PROGRAM CraneControl
VAR
	fbControlBox : FB_ControlBox; 
 	fbStatus : FB_Status;
	fbManualControl : FB_ManualControl; 
	bEnableManualControl : BOOL;
	fbAutomaticControl : FB_AutomaticControl;
	bEnableAutomaticControl : BOOL; 
	bEnableVFF : BOOL;
	bEnablePFC : BOOL;
	bEneableIC : BOOL;
	bEnableAD : BOOL;
	
	fOutManualTest : LREAL; 
	fOutAutomaticTest : LREAL;
END_VAR

fbControlBox(bRealControlBox := FALSE);

IF VirtualControlBox.stVirtualInputs.bOnSelector AND NOT(VirtualControlBox.stVirtualInputs.bAutoSelector) THEN
	bEnableManualControl := TRUE;	
ELSE
	bEnableManualControl := FALSE;
END_IF

fbManualControl(
	bEnable := bEnableManualControl,
	stParam := Parameters.stParam, 
	fVelocityFeedForwardControlOutput => fOutManualTest
);

IF VirtualControlBox.stVirtualInputs.bOnSelector AND VirtualControlBox.stVirtualInputs.bAutoSelector THEN
	bEnableAutomaticControl := TRUE;	
ELSE
	bEnableAutomaticControl := FALSE;
END_IF

fbAutomaticControl(
bEnable := bEnableAutomaticControl,
bEnableVelocityFeedForwardControl := bEnableVFF,
bEnableClosedLoopPositionControl := bEnablePFC,
bEnableIntegralController := bEneableIC,
bEnableActiveDamping := bEnableAD,
bActivateMotion := VirtualControlBox.stVirtualInputs.bStartButton,
bStopMotion := VirtualControlBox.stVirtualInputs.bStopButton,
stMotionReferenceGeneratorSettings := Parameters.stParam.stMotionReferenceGeneratorSettings,
stParam := Parameters.stParam,
fControlOutputNormalized => fOutAutomaticTest
);

END_PROGRAM

(* stored: Version 1.1.0.1, ProductVersion 3.1.4024.10
   POU CraneControl: Id {c8d14843-0c4e-4243-a583-0726f2828bd5}, SpecialFunc None *)
